(* IEC 61131-3 sources: TIAI/Course_examples/Carrello automatico/2020/build, 2 files *)

(* ---- plc.st ---- *)
TYPE
  LOGLEVEL : (CRITICAL, WARNING, INFO, DEBUG) := INFO;
END_TYPE

FUNCTION_BLOCK LOGGER
  VAR_INPUT
    TRIG : BOOL;
    MSG : STRING;
    LEVEL : LOGLEVEL := INFO;
  END_VAR
  VAR
    TRIG0 : BOOL;
  END_VAR

  IF TRIG AND NOT TRIG0 THEN
  {{
   LogMessage(GetFbVar(LEVEL),(char*)GetFbVar(MSG, .body),GetFbVar(MSG, .len));
  }}
  END_IF;
  TRIG0:=TRIG;
END_FUNCTION_BLOCK

FUNCTION_BLOCK python_eval
  VAR_INPUT
    TRIG : BOOL;
    CODE : STRING;
  END_VAR
  VAR_OUTPUT
    ACK : BOOL;
    RESULT : STRING;
  END_VAR
  VAR
    STATE : DWORD;
    BUFFER : STRING;
    PREBUFFER : STRING;
    TRIGM1 : BOOL;
    TRIGGED : BOOL;
  END_VAR

  {extern void __PythonEvalFB(int, PYTHON_EVAL*);__PythonEvalFB(0, data__);}
END_FUNCTION_BLOCK

FUNCTION_BLOCK python_poll
  VAR_INPUT
    TRIG : BOOL;
    CODE : STRING;
  END_VAR
  VAR_OUTPUT
    ACK : BOOL;
    RESULT : STRING;
  END_VAR
  VAR
    STATE : DWORD;
    BUFFER : STRING;
    PREBUFFER : STRING;
    TRIGM1 : BOOL;
    TRIGGED : BOOL;
  END_VAR

  {extern void __PythonEvalFB(int, PYTHON_EVAL*);__PythonEvalFB(1,(PYTHON_EVAL*)(void*)data__);}
END_FUNCTION_BLOCK

FUNCTION_BLOCK python_gear
  VAR_INPUT
    N : UINT;
    TRIG : BOOL;
    CODE : STRING;
  END_VAR
  VAR_OUTPUT
    ACK : BOOL;
    RESULT : STRING;
  END_VAR
  VAR
    py_eval : python_eval;
    COUNTER : UINT;
    ADD10_OUT : UINT;
    EQ13_OUT : BOOL;
    SEL15_OUT : UINT;
    AND7_OUT : BOOL;
  END_VAR

  ADD10_OUT := ADD(COUNTER, 1);
  EQ13_OUT := EQ(N, ADD10_OUT);
  SEL15_OUT := SEL(EQ13_OUT, ADD10_OUT, 0);
  COUNTER := SEL15_OUT;
  AND7_OUT := AND(EQ13_OUT, TRIG);
  py_eval(TRIG := AND7_OUT, CODE := CODE);
  ACK := py_eval.ACK;
  RESULT := py_eval.RESULT;
END_FUNCTION_BLOCK

PROGRAM main_carrello
  VAR
    g : BOOL := 0;
    fd : BOOL := 0;
    fs : BOOL := 0;
    fr : BOOL := 0;
    DX : BOOL := 0;
    SER : BOOL := 0;
    SX : BOOL := 0;
  END_VAR

  INITIAL_STEP quiete:
  END_STEP

  TRANSITION FROM quiete TO vai_a_dx
    := g;
  END_TRANSITION

  STEP vai_a_dx:
    DX(N);
  END_STEP

  TRANSITION FROM vai_a_dx TO carica
    := fd;
  END_TRANSITION

  STEP carica:
    SER(N);
  END_STEP

  TRANSITION FROM carica TO vai_a_sx
    := fr;
  END_TRANSITION

  STEP vai_a_sx:
    SX(N);
  END_STEP

  TRANSITION FROM vai_a_sx TO quiete
    := fs;
  END_TRANSITION

END_PROGRAM

CONFIGURATION Config0

  RESOURCE Res0 ON PLC
    TASK task0(INTERVAL := T#20ms,PRIORITY := 0);
    PROGRAM instance0 WITH task0 : main_carrello;
  END_RESOURCE
END_CONFIGURATION

(* ---- generated_plc.st ---- *)
PROGRAM main_carrello
  VAR
    g : BOOL := 0;
    fd : BOOL := 0;
    fs : BOOL := 0;
    fr : BOOL := 0;
    DX : BOOL := 0;
    SER : BOOL := 0;
    SX : BOOL := 0;
  END_VAR

  INITIAL_STEP quiete:
  END_STEP

  TRANSITION FROM quiete TO vai_a_dx
    := g;
  END_TRANSITION

  STEP vai_a_dx:
    DX(N);
  END_STEP

  TRANSITION FROM vai_a_dx TO carica
    := fd;
  END_TRANSITION

  STEP carica:
    SER(N);
  END_STEP

  TRANSITION FROM carica TO vai_a_sx
    := fr;
  END_TRANSITION

  STEP vai_a_sx:
    SX(N);
  END_STEP

  TRANSITION FROM vai_a_sx TO quiete
    := fs;
  END_TRANSITION

END_PROGRAM

CONFIGURATION Config0

  RESOURCE Res0 ON PLC
    TASK task0(INTERVAL := T#20ms,PRIORITY := 0);
    PROGRAM instance0 WITH task0 : main_carrello;
  END_RESOURCE
END_CONFIGURATION
